// TwinCAT 3 PLC project cvmi_motion
// ProgramVersion: 3.1.4026.15
// libraries:
//   LCLS General, * (SLAC)
//   Tc2_MC2, * (Beckhoff Automation GmbH)
//   Tc2_Standard, * (Beckhoff Automation GmbH)
//   Tc2_System, * (Beckhoff Automation GmbH)
//   Tc2_Utilities, * (Beckhoff Automation GmbH)
//   Tc3_Module, * (Beckhoff Automation GmbH)
//   lcls-twincat-motion,newest,SLAC
// project tree:
//   / PlcTask.TcTTO (not stored)
//   POUs/ Main.TcPOU
// real-time tasks:
//   TASK PlcTask: cycle T#10ms, priority 20, ADS port 350
// motion (NC):
//   TASK NC-Task 1 SAF: cycle T#2ms, priority 4, ADS port 501
//   TASK NC-Task 1 SVB: cycle T#10ms, priority 8, ADS port 511
//   AXIS GasJetX (id 1)
//     Dynamic: Acceleration=2, Deceleration=2, DelayTime=0.008
//     Velo: Maximum=1
//     TargetPosControl: Range=0.01, Time=0.1
//     OtherSettings: AllowMotionCmdToSlave=true
//     encoder EncType=4
//       EncPara: ScaleFactorNumerator=7.8125e-05, Inverse=true, MaxCount=#x0000ffff
//         SoftEndMaxControl: Range=16.1
//         Inc: RefSoftSyncMask=#x0000ffff
//     drive DrvType=24
//       DrvPara: Inverse=true
//         Analog: VeloReferenz=10, ScaleFactorActTorque=0.1
//         TimeComp: TaskDelayCycles=1
//     controller CtrType=1
//       CtrPara: PriorControlFactor=1
//         PosDiffControl: Range=0.5
//         Observer: BandWidth=20
//   AXIS GasJetY (id 2)
//     Dynamic: Acceleration=2, Deceleration=2, DelayTime=0.008
//     Velo: Maximum=1
//     TargetPosControl: Range=0.01, Time=0.1
//     OtherSettings: AllowMotionCmdToSlave=true
//     encoder EncType=4
//       EncPara: ScaleFactorNumerator=9.921875e-05, MaxCount=#x0000ffff
//         SoftEndMaxControl: Range=99.3
//         Inc: RefSoftSyncMask=#x0000ffff
//     drive DrvType=24
//       Analog: VeloReferenz=12.7, ScaleFactorActTorque=0.1
//       TimeComp: TaskDelayCycles=1
//     controller CtrType=1
//       CtrPara: PriorControlFactor=1
//         PosDiffControl: Range=0.5
//         Observer: BandWidth=20
//   AXIS GasJetZ (id 3)
//     Dynamic: Acceleration=2, Deceleration=2, DelayTime=0.008
//     Velo: Maximum=1
//     TargetPosControl: Range=0.01, Time=0.1
//     OtherSettings: AllowMotionCmdToSlave=true
//     encoder EncType=4
//       EncPara: ScaleFactorNumerator=8.59375e-05, MaxCount=#x0000ffff
//         SoftEndMaxControl: Range=29.4
//         Inc: RefSoftSyncMask=#x0000ffff
//     drive DrvType=24
//       Analog: VeloReferenz=11, ScaleFactorActTorque=0.1
//       TimeComp: TaskDelayCycles=1
//     controller CtrType=1
//       CtrPara: PriorControlFactor=1
//         PosDiffControl: Range=0.5
//         Observer: BandWidth=20
//   AXIS SamplePaddle (id 7)
//     General: UnitName=Degree
//     Dynamic: AccelerationMaximum=100, DecelerationMaximum=100, Acceleration=64.5934, Deceleration=64.5934, Jerk=417.23, DelayTime=0.008
//     Velo: Maximum=20
//     OtherSettings: AllowMotionCmdToSlave=true
//     encoder EncType=4
//       EncPara: ScaleFactorNumerator=0.0003125, Offset=-7.78125, MaxCount=#x0000ffff
//         SoftEndMinControl: Range=-2
//         SoftEndMaxControl: Range=2
//         Inc: RefSoftSyncMask=#x0000ffff
//     drive DrvType=24
//       Analog: VeloReferenz=10, ScaleFactorActTorque=0.1
//       TimeComp: TaskDelayCycles=1
//     controller CtrType=1
//       CtrPara: PriorControlFactor=1
//         PosDiffControl: Range=0.5
//         PID: PosKp=0
//         Observer: BandWidth=20
// I/O:
//   DEVICE Device 1 (EtherCAT), AmsNetId 172.21.68.243.2.1
//     Term 1 (EK1200) [EK1200-5000 EtherCAT Power supply (2A E-Bus)]
//       Term 2 (EL6070) [EL6070 1Ch. Licensing-Terminal]
//       EL7047-GasJet-X [EL7047 1Ch. Stepper motor output stage (50V, 5A)]
//       EL7047-GasJet-Y [EL7047 1Ch. Stepper motor output stage (50V, 5A)]
//       EL7047-GasJet-Z [EL7047 1Ch. Stepper motor output stage (50V, 5A)]
//       SamplePaddle-EL7047 [EL7047 1Ch. Stepper motor output stage (50V, 5A)]
//       Term 7 (EL7047) [EL7047 1Ch. Stepper motor output stage (50V, 5A)]
//       Term 8 (EL7047) [EL7047 1Ch. Stepper motor output stage (50V, 5A)]
//       Term 9 (EL9011) [EL9011 End Terminal]
// variable links:
//   (this object) <-> Device 1 (EtherCAT)/Term 1 (EK1200)/EL7047-GasJet-X
//     Drive/Inputs/In/nState1 @bit 3 <-> STM Status/Status/Error
//     Drive/Inputs/In/nState1 @bit 7 <-> STM Status/Status/Motor stall
//     Drive/Inputs/In/nState1 @bit 5 <-> STM Status/Status/Moving negative
//     Drive/Inputs/In/nState1 @bit 4 <-> STM Status/Status/Moving positive
//     Drive/Inputs/In/nState1 @bit 1 <-> STM Status/Status/Ready
//     Drive/Inputs/In/nState1 <-> STM Status/Status/Ready to enable
//     Drive/Inputs/In/nState1 @bit 6 <-> STM Status/Status/Torque reduced
//     Drive/Inputs/In/nState1 @bit 2 <-> STM Status/Status/Warning
//     Drive/Inputs/In/nState2 @bit 3 <-> STM Status/Status/Digital input 1
//     Drive/Inputs/In/nState2 @bit 4 <-> STM Status/Status/Digital input 2
//     Drive/Inputs/In/nState2 @bit 5 <-> STM Status/Status/Sync error
//     Drive/Inputs/In/nState2 @bit 7 <-> STM Status/Status/TxPDO Toggle
//     Drive/Inputs/In/nState4 @bit 1 <-> WcState/InputToggle
//     Drive/Inputs/In/nState4 <-> WcState/WcState
//     Drive/Outputs/Out/nCtrl1 <-> STM Control/Control/Enable
//     Drive/Outputs/Out/nCtrl1 @bit 2 <-> STM Control/Control/Reduce torque
//     Drive/Outputs/Out/nCtrl1 @bit 1 <-> STM Control/Control/Reset
//     Drive/Outputs/Out/nCtrl2 @bit 3 <-> STM Control/Control/Digital output 1
//     Drive/Outputs/Out/nDataOut2[0] <-> STM Velocity/Velocity
//     Enc/Inputs/In/nDataIn1[0] <-> ENC Status compact/Counter value
//     Enc/Inputs/In/nDataIn2[0] <-> ENC Status compact/Latch value
//     Enc/Inputs/In/nState1 @bit 4 <-> ENC Status compact/Status/Counter overflow
//     Enc/Inputs/In/nState1 @bit 3 <-> ENC Status compact/Status/Counter underflow
//     Enc/Inputs/In/nState1 @bit 7 <-> ENC Status compact/Status/Extrapolation stall
//     Enc/Inputs/In/nState1 <-> ENC Status compact/Status/Latch C valid
//     Enc/Inputs/In/nState1 @bit 1 <-> ENC Status compact/Status/Latch extern valid
//     Enc/Inputs/In/nState1 @bit 2 <-> ENC Status compact/Status/Set counter done
//     Enc/Inputs/In/nState2 @bit 4 <-> ENC Status compact/Status/Status of extern latch
//     Enc/Inputs/In/nState2 <-> ENC Status compact/Status/Status of input A
//     Enc/Inputs/In/nState2 @bit 1 <-> ENC Status compact/Status/Status of input B
//     Enc/Inputs/In/nState2 @bit 2 <-> ENC Status compact/Status/Status of input C
//     Enc/Inputs/In/nState2 @bit 5 <-> ENC Status compact/Status/Sync error
//     Enc/Inputs/In/nState2 @bit 7 <-> ENC Status compact/Status/TxPDO Toggle
//     Enc/Inputs/In/nState4 @bit 1 <-> WcState/InputToggle
//     Enc/Inputs/In/nState4 <-> WcState/WcState
//     Enc/Outputs/Out/nCtrl1 <-> ENC Control compact/Control/Enable latch C
//     Enc/Outputs/Out/nCtrl1 @bit 3 <-> ENC Control compact/Control/Enable latch extern on negative edge
//     Enc/Outputs/Out/nCtrl1 @bit 1 <-> ENC Control compact/Control/Enable latch extern on positive edge
//     Enc/Outputs/Out/nCtrl1 @bit 2 <-> ENC Control compact/Control/Set counter
//     Enc/Outputs/Out/nDataOut1[0] <-> ENC Control compact/Set counter value
//   (this object) <-> Device 1 (EtherCAT)/Term 1 (EK1200)/EL7047-GasJet-Y
//     Enc/Inputs/In/nDataIn1[0] <-> ENC Status compact/Counter value
//     Enc/Inputs/In/nDataIn2[0] <-> ENC Status compact/Latch value
//     Enc/Inputs/In/nState1 @bit 4 <-> ENC Status compact/Status/Counter overflow
//     Enc/Inputs/In/nState1 @bit 3 <-> ENC Status compact/Status/Counter underflow
//     Enc/Inputs/In/nState1 @bit 7 <-> ENC Status compact/Status/Extrapolation stall
//     Enc/Inputs/In/nState1 <-> ENC Status compact/Status/Latch C valid
//     Enc/Inputs/In/nState1 @bit 1 <-> ENC Status compact/Status/Latch extern valid
//     Enc/Inputs/In/nState1 @bit 2 <-> ENC Status compact/Status/Set counter done
//     Enc/Inputs/In/nState2 @bit 4 <-> ENC Status compact/Status/Status of extern latch
//     Enc/Inputs/In/nState2 <-> ENC Status compact/Status/Status of input A
//     Enc/Inputs/In/nState2 @bit 1 <-> ENC Status compact/Status/Status of input B
//     Enc/Inputs/In/nState2 @bit 2 <-> ENC Status compact/Status/Status of input C
//     Enc/Inputs/In/nState2 @bit 5 <-> ENC Status compact/Status/Sync error
//     Enc/Inputs/In/nState2 @bit 7 <-> ENC Status compact/Status/TxPDO Toggle
//     Enc/Inputs/In/nState4 @bit 1 <-> WcState/InputToggle
//     Enc/Inputs/In/nState4 <-> WcState/WcState
//     Enc/Outputs/Out/nCtrl1 <-> ENC Control compact/Control/Enable latch C
//     Enc/Outputs/Out/nCtrl1 @bit 3 <-> ENC Control compact/Control/Enable latch extern on negative edge
//     Enc/Outputs/Out/nCtrl1 @bit 1 <-> ENC Control compact/Control/Enable latch extern on positive edge
//     Enc/Outputs/Out/nCtrl1 @bit 2 <-> ENC Control compact/Control/Set counter
//     Enc/Outputs/Out/nDataOut1[0] <-> ENC Control compact/Set counter value
//   (this object) <-> Device 1 (EtherCAT)/Term 1 (EK1200)/EL7047-GasJet-Z
//     Drive/Inputs/In/nState1 @bit 3 <-> STM Status/Status/Error
//     Drive/Inputs/In/nState1 @bit 7 <-> STM Status/Status/Motor stall
//     Drive/Inputs/In/nState1 @bit 5 <-> STM Status/Status/Moving negative
//     Drive/Inputs/In/nState1 @bit 4 <-> STM Status/Status/Moving positive
//     Drive/Inputs/In/nState1 @bit 1 <-> STM Status/Status/Ready
//     Drive/Inputs/In/nState1 <-> STM Status/Status/Ready to enable
//     Drive/Inputs/In/nState1 @bit 6 <-> STM Status/Status/Torque reduced
//     Drive/Inputs/In/nState1 @bit 2 <-> STM Status/Status/Warning
//     Drive/Inputs/In/nState2 @bit 3 <-> STM Status/Status/Digital input 1
//     Drive/Inputs/In/nState2 @bit 4 <-> STM Status/Status/Digital input 2
//     Drive/Inputs/In/nState2 @bit 5 <-> STM Status/Status/Sync error
//     Drive/Inputs/In/nState2 @bit 7 <-> STM Status/Status/TxPDO Toggle
//     Drive/Inputs/In/nState4 @bit 1 <-> WcState/InputToggle
//     Drive/Inputs/In/nState4 <-> WcState/WcState
//     Drive/Outputs/Out/nCtrl1 <-> STM Control/Control/Enable
//     Drive/Outputs/Out/nCtrl1 @bit 2 <-> STM Control/Control/Reduce torque
//     Drive/Outputs/Out/nCtrl1 @bit 1 <-> STM Control/Control/Reset
//     Drive/Outputs/Out/nCtrl2 @bit 3 <-> STM Control/Control/Digital output 1
//     Drive/Outputs/Out/nDataOut2[0] <-> STM Velocity/Velocity
//     Enc/Inputs/In/nDataIn1[0] <-> ENC Status compact/Counter value
//     Enc/Inputs/In/nDataIn2[0] <-> ENC Status compact/Latch value
//     Enc/Inputs/In/nState1 @bit 4 <-> ENC Status compact/Status/Counter overflow
//     Enc/Inputs/In/nState1 @bit 3 <-> ENC Status compact/Status/Counter underflow
//     Enc/Inputs/In/nState1 @bit 7 <-> ENC Status compact/Status/Extrapolation stall
//     Enc/Inputs/In/nState1 <-> ENC Status compact/Status/Latch C valid
//     Enc/Inputs/In/nState1 @bit 1 <-> ENC Status compact/Status/Latch extern valid
//     Enc/Inputs/In/nState1 @bit 2 <-> ENC Status compact/Status/Set counter done
//     Enc/Inputs/In/nState2 @bit 4 <-> ENC Status compact/Status/Status of extern latch
//     Enc/Inputs/In/nState2 <-> ENC Status compact/Status/Status of input A
//     Enc/Inputs/In/nState2 @bit 1 <-> ENC Status compact/Status/Status of input B
//     Enc/Inputs/In/nState2 @bit 2 <-> ENC Status compact/Status/Status of input C
//     Enc/Inputs/In/nState2 @bit 5 <-> ENC Status compact/Status/Sync error
//     Enc/Inputs/In/nState2 @bit 7 <-> ENC Status compact/Status/TxPDO Toggle
//     Enc/Inputs/In/nState4 @bit 1 <-> WcState/InputToggle
//     Enc/Inputs/In/nState4 <-> WcState/WcState
//     Enc/Outputs/Out/nCtrl1 <-> ENC Control compact/Control/Enable latch C
//     Enc/Outputs/Out/nCtrl1 @bit 3 <-> ENC Control compact/Control/Enable latch extern on negative edge
//     Enc/Outputs/Out/nCtrl1 @bit 1 <-> ENC Control compact/Control/Enable latch extern on positive edge
//     Enc/Outputs/Out/nCtrl1 @bit 2 <-> ENC Control compact/Control/Set counter
//     Enc/Outputs/Out/nDataOut1[0] <-> ENC Control compact/Set counter value
//   (this object) <-> Device 1 (EtherCAT)/Term 1 (EK1200)/SamplePaddle-EL7047
//     Enc/Inputs/In/nDataIn1[0] <-> ENC Status compact/Counter value
//     Enc/Inputs/In/nDataIn2[0] <-> ENC Status compact/Latch value
//     Enc/Inputs/In/nState1 @bit 4 <-> ENC Status compact/Status/Counter overflow
//     Enc/Inputs/In/nState1 @bit 3 <-> ENC Status compact/Status/Counter underflow
//     Enc/Inputs/In/nState1 @bit 7 <-> ENC Status compact/Status/Extrapolation stall
//     Enc/Inputs/In/nState1 <-> ENC Status compact/Status/Latch C valid
//     Enc/Inputs/In/nState1 @bit 1 <-> ENC Status compact/Status/Latch extern valid
//     Enc/Inputs/In/nState1 @bit 2 <-> ENC Status compact/Status/Set counter done
//     Enc/Inputs/In/nState2 @bit 4 <-> ENC Status compact/Status/Status of extern latch
//     Enc/Inputs/In/nState2 <-> ENC Status compact/Status/Status of input A
//     Enc/Inputs/In/nState2 @bit 1 <-> ENC Status compact/Status/Status of input B
//     Enc/Inputs/In/nState2 @bit 2 <-> ENC Status compact/Status/Status of input C
//     Enc/Inputs/In/nState2 @bit 5 <-> ENC Status compact/Status/Sync error
//     Enc/Inputs/In/nState2 @bit 7 <-> ENC Status compact/Status/TxPDO Toggle
//     Enc/Inputs/In/nState4 @bit 1 <-> WcState/InputToggle
//     Enc/Inputs/In/nState4 <-> WcState/WcState
//     Enc/Outputs/Out/nCtrl1 <-> ENC Control compact/Control/Enable latch C
//     Enc/Outputs/Out/nCtrl1 @bit 3 <-> ENC Control compact/Control/Enable latch extern on negative edge
//     Enc/Outputs/Out/nCtrl1 @bit 1 <-> ENC Control compact/Control/Enable latch extern on positive edge
//     Enc/Outputs/Out/nCtrl1 @bit 2 <-> ENC Control compact/Control/Set counter
//     Enc/Outputs/Out/nDataOut1[0] <-> ENC Control compact/Set counter value
//   cvmi_motion Instance <-> Device 1 (EtherCAT)/Term 1 (EK1200)/EL7047-GasJet-X
//     PlcTask Inputs/Main.M1.bLimitBackwardEnable <-> STM Status/Status/Digital input 2
//     PlcTask Inputs/Main.M1.bLimitForwardEnable <-> STM Status/Status/Digital input 1
//   cvmi_motion Instance <-> Device 1 (EtherCAT)/Term 1 (EK1200)/EL7047-GasJet-Y
//     PlcTask Inputs/Main.M2.bLimitBackwardEnable <-> STM Status/Status/Digital input 2
//     PlcTask Inputs/Main.M2.bLimitForwardEnable <-> STM Status/Status/Digital input 1
//   cvmi_motion Instance <-> Device 1 (EtherCAT)/Term 1 (EK1200)/EL7047-GasJet-Z
//     PlcTask Inputs/Main.M3.bLimitBackwardEnable <-> STM Status/Status/Digital input 2
//     PlcTask Inputs/Main.M3.bLimitForwardEnable <-> STM Status/Status/Digital input 1
//   cvmi_motion Instance <-> Device 1 (EtherCAT)/Term 1 (EK1200)/SamplePaddle-EL7047
//     PlcTask Inputs/Main.M4.bLimitBackwardEnable <-> STM Status/Status/Digital input 2
//     PlcTask Inputs/Main.M4.bLimitForwardEnable <-> STM Status/Status/Digital input 1
//   cvmi_motion Instance <-> NC-Task 1 SAF/Axes/GasJetX
//     PlcTask Inputs/Main.M1.Axis.NcToPlc <-> Outputs/ToPlc
//     PlcTask Outputs/Main.M1.Axis.PlcToNc <-> Inputs/FromPlc
//   cvmi_motion Instance <-> NC-Task 1 SAF/Axes/GasJetY
//     PlcTask Inputs/Main.M2.Axis.NcToPlc <-> Outputs/ToPlc
//     PlcTask Outputs/Main.M2.Axis.PlcToNc <-> Inputs/FromPlc
//   cvmi_motion Instance <-> NC-Task 1 SAF/Axes/GasJetZ
//     PlcTask Inputs/Main.M3.Axis.NcToPlc <-> Outputs/ToPlc
//     PlcTask Outputs/Main.M3.Axis.PlcToNc <-> Inputs/FromPlc
//   cvmi_motion Instance <-> NC-Task 1 SAF/Axes/SamplePaddle
//     PlcTask Inputs/Main.M4.Axis.NcToPlc <-> Outputs/ToPlc
//     PlcTask Outputs/Main.M4.Axis.PlcToNc <-> Inputs/FromPlc

// ---- POUs/Main.TcPOU
PROGRAM Main
VAR
    // Motors
    // CVMI Axes
    {attribute 'TcLinkTo' := '.bLimitForwardEnable:=TIIB[EL7047-GasJet-X]^STM Status^Status^Digital input 1;    
                              .bLimitBackwardEnable:=TIIB[EL7047-GasJet-X]^STM Status^Status^Digital input 2'}
    {attribute 'pytmc' := '
        pv: CXI:CVMI:MMS:01
    '}
    M1 : ST_MotionStage := (bPowerSelf:=TRUE,
    nEnableMode:=ENUM_StageEnableMode.DURING_MOTION,
//    nEnableMode:=ENUM_StageEnableMode.ALWAYS,
    nHomingMode := ENUM_EpicsHomeCmd.ABSOLUTE_SET); // Gas Jet X

    {attribute 'TcLinkTo' := '.bLimitForwardEnable:=TIIB[EL7047-GasJet-Y]^STM Status^Status^Digital input 1;
                              .bLimitBackwardEnable:=TIIB[EL7047-GasJet-Y]^STM Status^Status^Digital input 2'}
    {attribute 'pytmc' := '
        pv: CXI:CVMI:MMS:02
    '}
    M2 : ST_MotionStage := (bPowerSelf:=TRUE,
    nEnableMode:=ENUM_StageEnableMode.DURING_MOTION,
//    nEnableMode:=ENUM_StageEnableMode.ALWAYS,
    nHomingMode := ENUM_EpicsHomeCmd.ABSOLUTE_SET); // Gas Jet Y

    {attribute 'TcLinkTo' := '.bLimitForwardEnable:=TIIB[EL7047-GasJet-Z]^STM Status^Status^Digital input 1;
                              .bLimitBackwardEnable:=TIIB[EL7047-GasJet-Z]^STM Status^Status^Digital input 2'}
    {attribute 'pytmc' := '
        pv: CXI:CVMI:MMS:03
    '}
    M3 : ST_MotionStage := (bPowerSelf:=TRUE,
    nEnableMode:=ENUM_StageEnableMode.DURING_MOTION,
//    nEnableMode:=ENUM_StageEnableMode.ALWAYS,
    nHomingMode := ENUM_EpicsHomeCmd.ABSOLUTE_SET); // Gas Jet Z


    {attribute 'TcLinkTo' := '.bLimitForwardEnable:=TIIB[SamplePaddle-EL7047]^STM Status^Status^Digital input 1;
                              .bLimitBackwardEnable:=TIIB[SamplePaddle-EL7047]^STM Status^Status^Digital input 2'}
    {attribute 'pytmc' := '
        pv: CXI:CVMI:MMS:04
    '}
    M4 : ST_MotionStage := (bPowerSelf:=TRUE,
    nEnableMode:=ENUM_StageEnableMode.DURING_MOTION,
//    nEnableMode:=ENUM_StageEnableMode.ALWAYS,
    nHomingMode := ENUM_EpicsHomeCmd.ABSOLUTE_SET); // Sample Paddle



    // CVMI Axes
    fbMotionStageM1 : FB_MotionStage;
    fbMotionStageM2 : FB_MotionStage;
    fbMotionStageM3 : FB_MotionStage;
    fbMotionStageM4 : FB_MotionStage;
END_VAR

    // Hardware Enable
    // CVMI
    // Gas Jet
    M1.bHardwareEnable := TRUE;
    M2.bHardwareEnable := TRUE;
    M3.bHardwareEnable := TRUE;
    // Gas Needle
    M4.bHardwareEnable := TRUE;



    // fbMotionStage
    // CVMI
    // Gas Jet
    fbMotionStageM1(stMotionStage:=M1);
    fbMotionStageM2(stMotionStage:=M2);
    fbMotionStageM3(stMotionStage:=M3);
    // Gas Needle
    fbMotionStageM4(stMotionStage:=M4);

END_PROGRAM
